TYPE U_Arrays3DimInOne :

UNION
	nData	: ARRAY[1..nMaxReadDataArray_3Dim] OF BYTE;
	bBool	: ARRAY[1..nArrayTestLength_3DimX, 1..nArrayTestLength_3DimY, 1..nArrayTestLength_3DimZ] OF BOOL;
	bByte	: ARRAY[1..nArrayTestLength_3DimX, 1..nArrayTestLength_3DimY, 1..nArrayTestLength_3DimZ] OF BYTE;
	nInt	: ARRAY[1..nArrayTestLength_3DimX, 1..nArrayTestLength_3DimY, 1..nArrayTestLength_3DimZ] OF INT;
	nUdint	: ARRAY[1..nArrayTestLength_3DimX, 1..nArrayTestLength_3DimY, 1..nArrayTestLength_3DimZ] OF UDINT;
	nReal	: ARRAY[1..nArrayTestLength_3DimX, 1..nArrayTestLength_3DimY, 1..nArrayTestLength_3DimZ] OF REAL;
	nLReal	: ARRAY[1..nArrayTestLength_3DimX, 1..nArrayTestLength_3DimY, 1..nArrayTestLength_3DimZ] OF LREAL;
	sString	: ARRAY[1..nArrayTestLength_3DimX, 1..nArrayTestLength_3DimY, 1..nArrayTestLength_3DimZ] OF STRING(80);
	wLword	: ARRAY[1..nArrayTestLength_3DimX, 1..nArrayTestLength_3DimY, 1..nArrayTestLength_3DimZ] OF LWORD;
	dDate	: ARRAY[1..nArrayTestLength_3DimX, 1..nArrayTestLength_3DimY, 1..nArrayTestLength_3DimZ] OF DT;
END_UNION

END_TYPE

(* stored: Version 1.1.0.1, ProductVersion 3.1.0.24
   DUT U_Arrays3DimInOne: Id {dd0fd11f-3d7a-41f8-aa91-d3eff1f45e21} *)
